(* PLC project MTCS, Beckhoff Automation GmbH TwinCAT PLC Control 3.5.13.21 *)
(* stored: creationDateTime 2024-06-13T11:53:15.8279126, modificationDateTime 2024-06-13T11:53:15.8279126 *)

FUNCTION_BLOCK SM_Pressure
VAR_INPUT
	///New pressure in Bar
	{attribute 'OPC.UA.DA' := '0'}
	newBarValue: LREAL;
END_VAR
VAR_OUTPUT
	///Current status description
	{attribute 'OPC.UA.DA' := '1'}
	{attribute 'OPC.UA.DA.Access' := '1'}
	actualStatus: STRING;
	///Previous status description
	previousStatus: STRING;
	///Pressure in Bar
	{attribute 'OPC.UA.DA' := '1'}
	{attribute 'OPC.UA.DA.Access' := '1'}
	bar: QuantityValue;
	///Pressure in Pascal
	{attribute 'OPC.UA.DA' := '1'}
	{attribute 'OPC.UA.DA.Access' := '1'}
	pascal: QuantityValue;
	///Pressure in HectoPascal
	{attribute 'OPC.UA.DA' := '1'}
	{attribute 'OPC.UA.DA.Access' := '1'}
	hectoPascal: QuantityValue;
END_VAR
VAR_IN_OUT
END_VAR
VAR
END_VAR

            bar(
    value := newBarValue,
    unit := Units.BAR);
pascal(
    value := newBarValue * 100000.0,
    unit := Units.PASCAL);

          

{attribute 'TcRpcEnable' := '1'}
METHOD _log : BOOL
VAR_INPUT
	///Name of this function block instance
	name: STRING;
END_VAR
VAR_OUTPUT
END_VAR
VAR_IN_OUT
	///Buffer to write all logging to
	buffer: LogBuffer;
END_VAR
VAR
	///Temporary buffer to write logging by parts (sub-statemachines) to
	subBuffer: LogBuffer;
END_VAR
                  LOGGER(
    name := name,
    actualStatus := THIS^.actualStatus,
    previousStatus := THIS^.previousStatus,
    buffer := buffer,
    subBuffer := subBuffer);

                
END_METHOD
END_FUNCTION_BLOCK
